// TIA Portal V21 export
TYPE "LBC_typeDigitalSignalConfiguration"
TITLE = LBC_typeDigitalSignalConfiguration
// Module related configuration parameters
   STRUCT
      referenceDesignator { S7_SetPoint := 'True'} : WString[25] := WSTRING#'DigitalSignal';   // Device name or device ID
      onDelay { S7_SetPoint := 'True'} : Time;   // Set time value for on delay
      offDelay { S7_SetPoint := 'True'} : Time;   // Set time value for off delay
      default { S7_SetPoint := 'True'} : Bool;   // Value to be returned if function block is not enabled or quality is bad (independent from `invertProcessValue`
      invertProcessValue { S7_SetPoint := 'True'} : Bool;   // Invert the process value (only the processed value, not the default)
      disableAlarms { S7_SetPoint := 'True'} : Bool;   // Disable the alarms of the block
   END_STRUCT;
END_TYPE
